Staubli VAL3: Robotscan.dtx

bool bSignal
bool bTxt1
bool bTxt2
bool bTxt3
bool btrig = true
public dio fout = {link=fOut0}
public frame FrmDraw = {x=1000, y=-100, fatherId=world[0]}
mdesc mNomSpeed
num l_nInit = 1500
num nNumTotal = 5031
num nNumrecord
public num nTranC[6]
num nTxtTotal = 11
num n_sTxt
num ndelay = 258.323
public num nnnn
num ntime = 459.89
pointRx pfrmCad[1500] = {fatherId=FrmDraw[0]}
public pointRx shere = {x=16.915, y=-25.265, z=273.2, rx=-177, ry=0.5, rz=-161.069, fatherId=FrmDraw[0]}
public sio sSocketout = {link=Socket\sSocketout}
string sString[1500]
tool tTool = {fatherId=flange[0], ioLink=valve1}
